PROGRAM NCI_MAIN
VAR 
 fbNci:FB_01_NCI;
 fbFalling :ARRAY[1..5] OF F_TRIG;
 fbRising  :ARRAY[1..5] OF R_TRIG;
 bEl5131_TrigH: BOOL;
 bEl5131_Trig : BOOL;
 bEl5131_TrigPressure: BOOL;
 tonWriteR:ARRAY [1..5] OF TON;
 bEl5131_ON :BOOL;
 stepWriteR:INT;
 
	tehn: INT;
END_VAR
VAR_IN_OUT
	
END_VAR

(*****************************************************************  
1.	out_stItpToPlc关联Channel2-inputs-FromPlc
    in_stItpToPlc 关联Channel2-output=ToPlc
2.  触发关联IO stIJP.bEx_TrigH/stIJP.bEx_Trig
*****************************************************************)
//底部真空破坏阀
IF Com_GVLS.bPlatformVacON THEN
	Y000002:=TRUE;
	Y000003:=FALSE;
END_IF

IF Com_GVLS.bPlatformVacOff THEN
	Y000002:=FALSE;
	Y000003:=TRUE;
END_IF

Y000001:=stIJP.bEx_TrigH OR bEl5131_TrigH  ;
Y000016:=(stIJP.bEx_Trig OR bEl5131_Trig )AND NOT stSystem.arErrorID[16];
stIJP.bEx_TrigHfb:=stIJP.bEx_TrigH OR bEl5131_TrigH ;

stIJP.bEx_Trigfb:=(stIJP.bEx_Trig OR bEl5131_Trig )AND NOT stSystem.arErrorID[16];
stIJP.bEx_TrigHfb:=stIJP.bEx_TrigH (*OR stIJP.bEl5131_Trig[1] OR stIJP_ZR.bEl5131_Trig *)(*AND  stSystem.arErrorID[15] AND   stSystem.arErrorID[16]
                      *)AND  stSystem.arErrorID[16];
stIJP.bEx_Trigfb:=(stIJP.bEx_Trig (*OR stIJP.bEl5131_Trig[1] OR stIJP_ZR.bEl5131_Trig *))(*AND  stSystem.arErrorID[15] AND   stSystem.arErrorID[16]
                      *)AND  stSystem.arErrorID[16];
					  
fbNci(
	stfbIJP:= stIJP, 
	in_stItpToPlc:= stIJP.in_stItpToPlc, 
	out_stItpToPlc:= stIJP.out_stItpToPlc, 
	nXAxisId:= arAXIS[1].NcToPlc.AxisId, 
	nYAxisId:= arAXIS[2].NcToPlc.AxisId, 
	nZAxisId:= arAXIS[4].NcToPlc.AxisId, 
	nQ1AxisId:= 0, 
	nQ2AxisId:= 0, 
	nChannelid:= stIJP.in_stItpToPlc.ChnId, 
	bProhibitMvALM:= );

IF stIJP.bStopExe THEN
   stIJP.bEx_TrigEl5131:=FALSE;
END_IF

// NCI报错监控 (error140-149)
stSystem.arErrorID[140+UDINT_TO_INT(stIJP.udiError)]:=stIJP.bError;

ACTION ACTNCIDispenser:
stIJP.strPRGName:=' 点胶XYZ插补';
stIJP.lrOverrideSet:=100;
(* IO关联*)
// NC:=stIJP.bEx_Trig;
stIJP.iJetOnDelay:=1;
END_ACTION

END_PROGRAM

(* stored: Version 1.1.0.1, ProductVersion 3.1.4024.12
   POU NCI_MAIN: Id {a95bee17-80a9-4312-9da1-6ab30ca06490}, SpecialFunc None
   Action ACTNCIDispenser: Id {6edf09c0-be99-437a-b9bd-38bbd4dba5cc} *)
